(* CODESYS project CoDeSys PLC Program-Client.project

Project tree, tasks and I/O mapping:
  Device : CECC-LK, Festo AG & Co. KG, order no. 574418, version 3.5.0.7
    application Application
      libraries: Util, 3.5.0.0 (System); OPAK_RFID, 3.5.0.0 (elrest Automationssysteme GmbH); Solution Center Library, 3.5.8.0 (Festo Didactic SE - Customer Solution Center); Network, 3.5.7.0 (3S - Smart Software Solutions GmbH); Standard, 3.5.9.0 (System); Solution Center Library, 3.5.8.0 (Festo Didactic SE - Customer Solution Center); CAA CiA 405, 3.5.0.0 (CAA Technical Workgroup)
      task MainTask (cyclic, interval t#20ms, priority 20) calls PLC_PRG
      program PLC_PRG [ST]
      global variables IO
    Onboard : CECC 14I/8O, Festo AG & Co. KG, version 3.4.5.5
        unmapped channels: Onboard Input, Onboard Output
      Digital Inputs
          unmapped channels: Onboard Input
      Digital Outputs
          unmapped channels: Onboard Output
    CAN : CANbus, 3S - Smart Software Solutions GmbH, version 3.5.7.0
        settings: Baudrate = 1000
      CANopen : CANopen_Manager, 3S - Smart Software Solutions GmbH, order no. 1806, version 3.5.0.0
          settings: Sync CycleTime in Microseconds = 8000; Synchronous Window Length = 0; Enable Heartbeat generation = FALSE; CANopen NodeID = 1; ConfigVersion = 50659328
        BL20_GWBR_CANOPEN : BL20-GWBR-CANOPEN, TURCK, order no. 6827167, version Revision=16#00040017, FileVersion=4.23
            settings: General Options.Reset Node = FALSE; NODEIDSAVED = 2; SDO Timeout = 1000000; EXPERTSETTINGS = TRUE; Emergency-General Parameters.Emergency COBID = 16#82; Settings.COBID = 16#00000202; Settings.Transmission Type = 16#FF; Settings.available PDO-Parameter.Inhibit Time available = FALSE; Settings.available PDO-Parameter.Event Timer available = FALSE; Settings.Inhibit Time = 0; Settings.Event Timer = 0; Generic COBID = '$NODEID+16#0200'; Process by CANopenManager = TRUE; Settings.COBID = 16#00000302; Settings.Transmission Type = 16#FF; Settings.available PDO-Parameter.Inhibit Time available = FALSE; Settings.available PDO-Parameter.Event Timer available = FALSE; Settings.Inhibit Time = 0; Settings.Event Timer = 0; Generic COBID = '$NODEID+16#0300'; Process by CANopenManager = TRUE; Settings.COBID = 16#00000182; Settings.Transmission Type = 16#FF; Settings.available PDO-Parameter.Inhibit Time available = TRUE; Settings.available PDO-Parameter.Event Timer available = TRUE; Settings.Inhibit Time = 0; Settings.Event Timer = 0; Generic COBID = '$NODEID+16#0180'; Process by CANopenManager = TRUE; Settings.COBID = 16#00000282; Settings.Transmission Type = 16#FF; Settings.available PDO-Parameter.Inhibit Time available = TRUE; Settings.available PDO-Parameter.Event Timer available = TRUE; Settings.Inhibit Time = 0; Settings.Event Timer = 0; Generic COBID = '$NODEID+16#0280'; Process by CANopenManager = TRUE; WriteOutput8Bit : Generic_BL20_4DO.Index = 16#6200; WriteOutput8Bit : Generic_BL20_4DO.Subindex = 16#01; WriteOutput8Bit : Generic_BL20_4DO.ObjectLength = 8;
              WriteOutput8Bit : Generic_BL20_4DO_2.Index = 16#6200; WriteOutput8Bit : Generic_BL20_4DO_2.Subindex = 16#02; WriteOutput8Bit : Generic_BL20_4DO_2.ObjectLength = 8; WriteAnalogueOutput16 : Generic_BL20_2AO.Index = 16#6411; WriteAnalogueOutput16 : Generic_BL20_2AO.Subindex = 16#01; WriteAnalogueOutput16 : Generic_BL20_2AO.ObjectLength = 16; WriteAnalogueOutput16 : Generic_BL20_2AO.Index = 16#6411; WriteAnalogueOutput16 : Generic_BL20_2AO.Subindex = 16#02; WriteAnalogueOutput16 : Generic_BL20_2AO.ObjectLength = 16; ReadInput8Bit : Generic_BL20_4DI.Index = 16#6000; ReadInput8Bit : Generic_BL20_4DI.Subindex = 16#01; ReadInput8Bit : Generic_BL20_4DI.ObjectLength = 8; ReadAnalogueInput16Bit : Generic_BL20_4AI.Index = 16#6401; ReadAnalogueInput16Bit : Generic_BL20_4AI.Subindex = 16#01; ReadAnalogueInput16Bit : Generic_BL20_4AI.ObjectLength = 16; ReadAnalogueInput16Bit : Generic_BL20_4AI.Index = 16#6401; ReadAnalogueInput16Bit : Generic_BL20_4AI.Subindex = 16#02; ReadAnalogueInput16Bit : Generic_BL20_4AI.ObjectLength = 16; ReadAnalogueInput16Bit : Generic_BL20_4AI.Index = 16#6401; ReadAnalogueInput16Bit : Generic_BL20_4AI.Subindex = 16#03; ReadAnalogueInput16Bit : Generic_BL20_4AI.ObjectLength = 16; ReadAnalogueInput16Bit : Generic_BL20_4AI.Index = 16#6401; ReadAnalogueInput16Bit : Generic_BL20_4AI.Subindex = 16#04; ReadAnalogueInput16Bit : Generic_BL20_4AI.ObjectLength = 16; Number of SDO = 39; Set Guardtime.Index = 16#100C; Set Guardtime.Subindex = 16#00; Set Guardtime.Value = 16#00000000; Set Guardtime.Size = 16; Set Guardtime.AbortIfError = FALSE; Set Guardtime.JumpToLine = FALSE; Set Guardtime.Line = 0; Set Lifetime.Index = 16#100D; Set Lifetime.Subindex = 16#00; Set Lifetime.Value = 16#00000000; Set Lifetime.Size = 8; Set Lifetime.AbortIfError = FALSE; Set Lifetime.JumpToLine = FALSE; Set Lifetime.Line = 0; Disable Emcy CobID.Index = 16#1014;
              Disable Emcy CobID.Subindex = 16#00; Disable Emcy CobID.Value = 16#80000082; Disable Emcy CobID.Size = 32; Disable Emcy CobID.AbortIfError = FALSE; Disable Emcy CobID.JumpToLine = FALSE; Disable Emcy CobID.Line = 0; Set Emcy CobID.Index = 16#1014; Set Emcy CobID.Subindex = 16#00; Set Emcy CobID.Value = 16#00000082; Set Emcy CobID.Size = 32; Set Emcy CobID.AbortIfError = FALSE; Set Emcy CobID.JumpToLine = FALSE; Set Emcy CobID.Line = 0; Set Heartbeat Consumer.Index = 16#1016; Set Heartbeat Consumer.Subindex = 16#01; Set Heartbeat Consumer.Value = 0; Set Heartbeat Consumer.Size = 32; Set Heartbeat Consumer.AbortIfError = FALSE; Set Heartbeat Consumer.JumpToLine = FALSE; Set Heartbeat Consumer.Line = 0; Set Heartbeat Producer.Index = 16#1017; Set Heartbeat Producer.Subindex = 16#00; Set Heartbeat Producer.Value = 16#00000000; Set Heartbeat Producer.Size = 16; Set Heartbeat Producer.AbortIfError = FALSE; Set Heartbeat Producer.JumpToLine = FALSE; Set Heartbeat Producer.Line = 0; Disable PDO.Index = 16#1400; Disable PDO.Subindex = 16#01; Disable PDO.Value = 16#80000202; Disable PDO.Size = 32; Disable PDO.AbortIfError = FALSE; Disable PDO.JumpToLine = FALSE; Disable PDO.Line = 0; Set transmission type.Index = 16#1400; Set transmission type.Subindex = 16#02; Set transmission type.Value = 16#FF; Set transmission type.Size = 8; Set transmission type.AbortIfError = FALSE; Set transmission type.JumpToLine = FALSE;
              Set transmission type.Line = 0; Clear pdo mapping.Index = 16#1600; Clear pdo mapping.Subindex = 16#00; Clear pdo mapping.Value = 16#0; Clear pdo mapping.Size = 8; Clear pdo mapping.AbortIfError = FALSE; Clear pdo mapping.JumpToLine = FALSE; Clear pdo mapping.Line = 0; Set Mapping.Index = 16#1600; Set Mapping.Subindex = 16#01; Set Mapping.Value = 16#62000108; Set Mapping.Size = 32; Set Mapping.AbortIfError = FALSE; Set Mapping.JumpToLine = FALSE; Set Mapping.Line = 0; Set Mapping.Index = 16#1600; Set Mapping.Subindex = 16#02; Set Mapping.Value = 16#62000208; Set Mapping.Size = 32; Set Mapping.AbortIfError = FALSE; Set Mapping.JumpToLine = FALSE; Set Mapping.Line = 0; Set number of mappings.Index = 16#1600; Set number of mappings.Subindex = 16#00; Set number of mappings.Value = 16#02; Set number of mappings.Size = 8; Set number of mappings.AbortIfError = FALSE; Set number of mappings.JumpToLine = FALSE; Set number of mappings.Line = 0; Set and enable COB-ID.Index = 16#1400; Set and enable COB-ID.Subindex = 16#01; Set and enable COB-ID.Value = 16#00000202; Set and enable COB-ID.Size = 32; Set and enable COB-ID.AbortIfError = FALSE; Set and enable COB-ID.JumpToLine = FALSE; Set and enable COB-ID.Line = 0; Disable PDO.Index = 16#1401; Disable PDO.Subindex = 16#01; Disable PDO.Value = 16#80000302; Disable PDO.Size = 32;
              Disable PDO.AbortIfError = FALSE; Disable PDO.JumpToLine = FALSE; Disable PDO.Line = 0; Set transmission type.Index = 16#1401; Set transmission type.Subindex = 16#02; Set transmission type.Value = 16#FF; Set transmission type.Size = 8; Set transmission type.AbortIfError = FALSE; Set transmission type.JumpToLine = FALSE; Set transmission type.Line = 0; Clear pdo mapping.Index = 16#1601; Clear pdo mapping.Subindex = 16#00; Clear pdo mapping.Value = 16#0; Clear pdo mapping.Size = 8; Clear pdo mapping.AbortIfError = FALSE; Clear pdo mapping.JumpToLine = FALSE; Clear pdo mapping.Line = 0; Set Mapping.Index = 16#1601; Set Mapping.Subindex = 16#01; Set Mapping.Value = 16#64110110; Set Mapping.Size = 32; Set Mapping.AbortIfError = FALSE; Set Mapping.JumpToLine = FALSE; Set Mapping.Line = 0; Set Mapping.Index = 16#1601; Set Mapping.Subindex = 16#02; Set Mapping.Value = 16#64110210; Set Mapping.Size = 32; Set Mapping.AbortIfError = FALSE; Set Mapping.JumpToLine = FALSE; Set Mapping.Line = 0; Set number of mappings.Index = 16#1601; Set number of mappings.Subindex = 16#00; Set number of mappings.Value = 16#02; Set number of mappings.Size = 8; Set number of mappings.AbortIfError = FALSE; Set number of mappings.JumpToLine = FALSE; Set number of mappings.Line = 0; Set and enable COB-ID.Index = 16#1401; Set and enable COB-ID.Subindex = 16#01;
              Set and enable COB-ID.Value = 16#00000302; Set and enable COB-ID.Size = 32; Set and enable COB-ID.AbortIfError = FALSE; Set and enable COB-ID.JumpToLine = FALSE; Set and enable COB-ID.Line = 0; Disable PDO.Index = 16#1800; Disable PDO.Subindex = 16#01; Disable PDO.Value = 16#80000182; Disable PDO.Size = 32; Disable PDO.AbortIfError = FALSE; Disable PDO.JumpToLine = FALSE; Disable PDO.Line = 0; Set transmission type.Index = 16#1800; Set transmission type.Subindex = 16#02; Set transmission type.Value = 16#FF; Set transmission type.Size = 8; Set transmission type.AbortIfError = FALSE; Set transmission type.JumpToLine = FALSE; Set transmission type.Line = 0; Set inhibit time.Index = 16#1800; Set inhibit time.Subindex = 16#03; Set inhibit time.Value = 16#0000; Set inhibit time.Size = 16; Set inhibit time.AbortIfError = FALSE; Set inhibit time.JumpToLine = FALSE; Set inhibit time.Line = 0; Set event time.Index = 16#1800; Set event time.Subindex = 16#05; Set event time.Value = 16#0000; Set event time.Size = 16; Set event time.AbortIfError = FALSE; Set event time.JumpToLine = FALSE; Set event time.Line = 0; Clear pdo mapping.Index = 16#1A00; Clear pdo mapping.Subindex = 16#00; Clear pdo mapping.Value = 16#0; Clear pdo mapping.Size = 8; Clear pdo mapping.AbortIfError = FALSE; Clear pdo mapping.JumpToLine = FALSE; Clear pdo mapping.Line = 0;
              Set Mapping.Index = 16#1A00; Set Mapping.Subindex = 16#01; Set Mapping.Value = 16#60000108; Set Mapping.Size = 32; Set Mapping.AbortIfError = FALSE; Set Mapping.JumpToLine = FALSE; Set Mapping.Line = 0; Set number of mappings.Index = 16#1A00; Set number of mappings.Subindex = 16#00; Set number of mappings.Value = 16#01; Set number of mappings.Size = 8; Set number of mappings.AbortIfError = FALSE; Set number of mappings.JumpToLine = FALSE; Set number of mappings.Line = 0; Set and enable COB-ID.Index = 16#1800; Set and enable COB-ID.Subindex = 16#01; Set and enable COB-ID.Value = 16#00000182; Set and enable COB-ID.Size = 32; Set and enable COB-ID.AbortIfError = FALSE; Set and enable COB-ID.JumpToLine = FALSE; Set and enable COB-ID.Line = 0; Disable PDO.Index = 16#1801; Disable PDO.Subindex = 16#01; Disable PDO.Value = 16#80000282; Disable PDO.Size = 32; Disable PDO.AbortIfError = FALSE; Disable PDO.JumpToLine = FALSE; Disable PDO.Line = 0; Set transmission type.Index = 16#1801; Set transmission type.Subindex = 16#02; Set transmission type.Value = 16#FF; Set transmission type.Size = 8; Set transmission type.AbortIfError = FALSE; Set transmission type.JumpToLine = FALSE; Set transmission type.Line = 0; Set inhibit time.Index = 16#1801; Set inhibit time.Subindex = 16#03; Set inhibit time.Value = 16#0000; Set inhibit time.Size = 16; Set inhibit time.AbortIfError = FALSE;
              Set inhibit time.JumpToLine = FALSE; Set inhibit time.Line = 0; Set event time.Index = 16#1801; Set event time.Subindex = 16#05; Set event time.Value = 16#0000; Set event time.Size = 16; Set event time.AbortIfError = FALSE; Set event time.JumpToLine = FALSE; Set event time.Line = 0; Clear pdo mapping.Index = 16#1A01; Clear pdo mapping.Subindex = 16#00; Clear pdo mapping.Value = 16#0; Clear pdo mapping.Size = 8; Clear pdo mapping.AbortIfError = FALSE; Clear pdo mapping.JumpToLine = FALSE; Clear pdo mapping.Line = 0; Set Mapping.Index = 16#1A01; Set Mapping.Subindex = 16#01; Set Mapping.Value = 16#64010110; Set Mapping.Size = 32; Set Mapping.AbortIfError = FALSE; Set Mapping.JumpToLine = FALSE; Set Mapping.Line = 0; Set Mapping.Index = 16#1A01; Set Mapping.Subindex = 16#02; Set Mapping.Value = 16#64010210; Set Mapping.Size = 32; Set Mapping.AbortIfError = FALSE; Set Mapping.JumpToLine = FALSE; Set Mapping.Line = 0; Set Mapping.Index = 16#1A01; Set Mapping.Subindex = 16#03; Set Mapping.Value = 16#64010310; Set Mapping.Size = 32; Set Mapping.AbortIfError = FALSE; Set Mapping.JumpToLine = FALSE; Set Mapping.Line = 0; Set Mapping.Index = 16#1A01; Set Mapping.Subindex = 16#04; Set Mapping.Value = 16#64010410;
              Set Mapping.Size = 32; Set Mapping.AbortIfError = FALSE; Set Mapping.JumpToLine = FALSE; Set Mapping.Line = 0; Set number of mappings.Index = 16#1A01; Set number of mappings.Subindex = 16#00; Set number of mappings.Value = 16#04; Set number of mappings.Size = 8; Set number of mappings.AbortIfError = FALSE; Set number of mappings.JumpToLine = FALSE; Set number of mappings.Line = 0; Set and enable COB-ID.Index = 16#1801; Set and enable COB-ID.Subindex = 16#01; Set and enable COB-ID.Value = 16#00000282; Set and enable COB-ID.Size = 32; Set and enable COB-ID.AbortIfError = FALSE; Set and enable COB-ID.JumpToLine = FALSE; Set and enable COB-ID.Line = 0; ConfigVersion = 50659328
          Generic_BL20_4DI : Generic BL20-4DI, TURCK, order no. 0, version Revision=16#00040017, FileVersion=4.23
              settings: Number of Params = 0; Number of Params = 4; ReadInput8Bit : Generic_BL20_4DI.Index = 16#6000; ReadInput8Bit : Generic_BL20_4DI.Subindex = 16#01; ReadInput8Bit : Generic_BL20_4DI.Startbit = 0; ReadInput8Bit : Generic_BL20_4DI.Endbit = 0; ReadInput8Bit : Generic_BL20_4DI.Index = 16#6000; ReadInput8Bit : Generic_BL20_4DI.Subindex = 16#01; ReadInput8Bit : Generic_BL20_4DI.Startbit = 1; ReadInput8Bit : Generic_BL20_4DI.Endbit = 1; ReadInput8Bit : Generic_BL20_4DI.Index = 16#6000; ReadInput8Bit : Generic_BL20_4DI.Subindex = 16#01; ReadInput8Bit : Generic_BL20_4DI.Startbit = 2; ReadInput8Bit : Generic_BL20_4DI.Endbit = 2; ReadInput8Bit : Generic_BL20_4DI.Index = 16#6000; ReadInput8Bit : Generic_BL20_4DI.Subindex = 16#01; ReadInput8Bit : Generic_BL20_4DI.Startbit = 3; ReadInput8Bit : Generic_BL20_4DI.Endbit = 3
              unmapped channels: ReadInput8Bit : Generic_BL20_4DI, ReadInput8Bit : Generic_BL20_4DI, ReadInput8Bit : Generic_BL20_4DI, ReadInput8Bit : Generic_BL20_4DI
          Generic_BL20_4DI_1 : Generic BL20-4DI, TURCK, order no. 0, version Revision=16#00040017, FileVersion=4.23
              settings: Number of Params = 0; Number of Params = 4; ReadInput8Bit : Generic_BL20_4DI.Index = 16#6000; ReadInput8Bit : Generic_BL20_4DI.Subindex = 16#01; ReadInput8Bit : Generic_BL20_4DI.Startbit = 4; ReadInput8Bit : Generic_BL20_4DI.Endbit = 4; ReadInput8Bit : Generic_BL20_4DI.Index = 16#6000; ReadInput8Bit : Generic_BL20_4DI.Subindex = 16#01; ReadInput8Bit : Generic_BL20_4DI.Startbit = 5; ReadInput8Bit : Generic_BL20_4DI.Endbit = 5; ReadInput8Bit : Generic_BL20_4DI.Index = 16#6000; ReadInput8Bit : Generic_BL20_4DI.Subindex = 16#01; ReadInput8Bit : Generic_BL20_4DI.Startbit = 6; ReadInput8Bit : Generic_BL20_4DI.Endbit = 6; ReadInput8Bit : Generic_BL20_4DI.Index = 16#6000; ReadInput8Bit : Generic_BL20_4DI.Subindex = 16#01; ReadInput8Bit : Generic_BL20_4DI.Startbit = 7; ReadInput8Bit : Generic_BL20_4DI.Endbit = 7
              unmapped channels: ReadInput8Bit : Generic_BL20_4DI, ReadInput8Bit : Generic_BL20_4DI, ReadInput8Bit : Generic_BL20_4DI, ReadInput8Bit : Generic_BL20_4DI
          Generic_BL20_BR_PF : Generic BL20-BR/-PF, TURCK, order no. 0, version Revision=16#00040017, FileVersion=4.23
              settings: Number of Params = 0; Number of Params = 0
          Generic_BL20_4DO : Generic BL20-4DO, TURCK, order no. 0, version Revision=16#00040017, FileVersion=4.23
              settings: Number of Params = 4; WriteOutput8Bit : Generic_BL20_4DO.Index = 16#6200; WriteOutput8Bit : Generic_BL20_4DO.Subindex = 16#01; WriteOutput8Bit : Generic_BL20_4DO.Startbit = 0; WriteOutput8Bit : Generic_BL20_4DO.Endbit = 0; WriteOutput8Bit : Generic_BL20_4DO.Index = 16#6200; WriteOutput8Bit : Generic_BL20_4DO.Subindex = 16#01; WriteOutput8Bit : Generic_BL20_4DO.Startbit = 1; WriteOutput8Bit : Generic_BL20_4DO.Endbit = 1; WriteOutput8Bit : Generic_BL20_4DO.Index = 16#6200; WriteOutput8Bit : Generic_BL20_4DO.Subindex = 16#01; WriteOutput8Bit : Generic_BL20_4DO.Startbit = 2; WriteOutput8Bit : Generic_BL20_4DO.Endbit = 2; WriteOutput8Bit : Generic_BL20_4DO.Index = 16#6200; WriteOutput8Bit : Generic_BL20_4DO.Subindex = 16#01; WriteOutput8Bit : Generic_BL20_4DO.Startbit = 3; WriteOutput8Bit : Generic_BL20_4DO.Endbit = 3; Number of Params = 0
              unmapped channels: WriteOutput8Bit : Generic_BL20_4DO, WriteOutput8Bit : Generic_BL20_4DO, WriteOutput8Bit : Generic_BL20_4DO, WriteOutput8Bit : Generic_BL20_4DO
          Generic_BL20_4DO_1 : Generic BL20-4DO, TURCK, order no. 0, version Revision=16#00040017, FileVersion=4.23
              settings: Number of Params = 4; WriteOutput8Bit : Generic_BL20_4DO.Index = 16#6200; WriteOutput8Bit : Generic_BL20_4DO.Subindex = 16#01; WriteOutput8Bit : Generic_BL20_4DO.Startbit = 4; WriteOutput8Bit : Generic_BL20_4DO.Endbit = 4; WriteOutput8Bit : Generic_BL20_4DO.Index = 16#6200; WriteOutput8Bit : Generic_BL20_4DO.Subindex = 16#01; WriteOutput8Bit : Generic_BL20_4DO.Startbit = 5; WriteOutput8Bit : Generic_BL20_4DO.Endbit = 5; WriteOutput8Bit : Generic_BL20_4DO.Index = 16#6200; WriteOutput8Bit : Generic_BL20_4DO.Subindex = 16#01; WriteOutput8Bit : Generic_BL20_4DO.Startbit = 6; WriteOutput8Bit : Generic_BL20_4DO.Endbit = 6; WriteOutput8Bit : Generic_BL20_4DO.Index = 16#6200; WriteOutput8Bit : Generic_BL20_4DO.Subindex = 16#01; WriteOutput8Bit : Generic_BL20_4DO.Startbit = 7; WriteOutput8Bit : Generic_BL20_4DO.Endbit = 7; Number of Params = 0
              unmapped channels: WriteOutput8Bit : Generic_BL20_4DO, WriteOutput8Bit : Generic_BL20_4DO, WriteOutput8Bit : Generic_BL20_4DO, WriteOutput8Bit : Generic_BL20_4DO
          Generic_BL20_4DO_2 : Generic BL20-4DO, TURCK, order no. 0, version Revision=16#00040017, FileVersion=4.23
              settings: Number of Params = 4; WriteOutput8Bit : Generic_BL20_4DO_2.Index = 16#6200; WriteOutput8Bit : Generic_BL20_4DO_2.Subindex = 16#02; WriteOutput8Bit : Generic_BL20_4DO_2.Startbit = 0; WriteOutput8Bit : Generic_BL20_4DO_2.Endbit = 0; WriteOutput8Bit : Generic_BL20_4DO_2.Index = 16#6200; WriteOutput8Bit : Generic_BL20_4DO_2.Subindex = 16#02; WriteOutput8Bit : Generic_BL20_4DO_2.Startbit = 1; WriteOutput8Bit : Generic_BL20_4DO_2.Endbit = 1; WriteOutput8Bit : Generic_BL20_4DO_2.Index = 16#6200; WriteOutput8Bit : Generic_BL20_4DO_2.Subindex = 16#02; WriteOutput8Bit : Generic_BL20_4DO_2.Startbit = 2; WriteOutput8Bit : Generic_BL20_4DO_2.Endbit = 2; WriteOutput8Bit : Generic_BL20_4DO_2.Index = 16#6200; WriteOutput8Bit : Generic_BL20_4DO_2.Subindex = 16#02; WriteOutput8Bit : Generic_BL20_4DO_2.Startbit = 3; WriteOutput8Bit : Generic_BL20_4DO_2.Endbit = 3; Number of Params = 0
              unmapped channels: WriteOutput8Bit : Generic_BL20_4DO_2, WriteOutput8Bit : Generic_BL20_4DO_2, WriteOutput8Bit : Generic_BL20_4DO_2, WriteOutput8Bit : Generic_BL20_4DO_2
          Generic_BL20_4DO_3 : Generic BL20-4DO, TURCK, order no. 0, version Revision=16#00040017, FileVersion=4.23
              settings: Number of Params = 4; WriteOutput8Bit : Generic_BL20_4DO_2.Index = 16#6200; WriteOutput8Bit : Generic_BL20_4DO_2.Subindex = 16#02; WriteOutput8Bit : Generic_BL20_4DO_2.Startbit = 4; WriteOutput8Bit : Generic_BL20_4DO_2.Endbit = 4; WriteOutput8Bit : Generic_BL20_4DO_2.Index = 16#6200; WriteOutput8Bit : Generic_BL20_4DO_2.Subindex = 16#02; WriteOutput8Bit : Generic_BL20_4DO_2.Startbit = 5; WriteOutput8Bit : Generic_BL20_4DO_2.Endbit = 5; WriteOutput8Bit : Generic_BL20_4DO_2.Index = 16#6200; WriteOutput8Bit : Generic_BL20_4DO_2.Subindex = 16#02; WriteOutput8Bit : Generic_BL20_4DO_2.Startbit = 6; WriteOutput8Bit : Generic_BL20_4DO_2.Endbit = 6; WriteOutput8Bit : Generic_BL20_4DO_2.Index = 16#6200; WriteOutput8Bit : Generic_BL20_4DO_2.Subindex = 16#02; WriteOutput8Bit : Generic_BL20_4DO_2.Startbit = 7; WriteOutput8Bit : Generic_BL20_4DO_2.Endbit = 7; Number of Params = 0
              unmapped channels: WriteOutput8Bit : Generic_BL20_4DO_2, WriteOutput8Bit : Generic_BL20_4DO_2, WriteOutput8Bit : Generic_BL20_4DO_2, WriteOutput8Bit : Generic_BL20_4DO_2
          Generic_BL20_2AO : Generic BL20-2AO, TURCK, order no. 0, version Revision=16#00040017, FileVersion=4.23
              settings: Number of Params = 2; WriteAnalogueOutput16 : Generic_BL20_2AO.Index = 16#6411; WriteAnalogueOutput16 : Generic_BL20_2AO.Subindex = 16#01; WriteAnalogueOutput16 : Generic_BL20_2AO.Startbit = 0; WriteAnalogueOutput16 : Generic_BL20_2AO.Endbit = 15; WriteAnalogueOutput16 : Generic_BL20_2AO.Index = 16#6411; WriteAnalogueOutput16 : Generic_BL20_2AO.Subindex = 16#02; WriteAnalogueOutput16 : Generic_BL20_2AO.Startbit = 0; WriteAnalogueOutput16 : Generic_BL20_2AO.Endbit = 15; Number of Params = 0
              unmapped channels: WriteAnalogueOutput16 : Generic_BL20_2AO, WriteAnalogueOutput16 : Generic_BL20_2AO
          Generic_BL20_4AI : Generic BL20-4AI, TURCK, order no. 0, version Revision=16#00040017, FileVersion=4.23
              settings: Number of Params = 0; Number of Params = 4; ReadAnalogueInput16Bit : Generic_BL20_4AI.Index = 16#6401; ReadAnalogueInput16Bit : Generic_BL20_4AI.Subindex = 16#01; ReadAnalogueInput16Bit : Generic_BL20_4AI.Startbit = 0; ReadAnalogueInput16Bit : Generic_BL20_4AI.Endbit = 15; ReadAnalogueInput16Bit : Generic_BL20_4AI.Index = 16#6401; ReadAnalogueInput16Bit : Generic_BL20_4AI.Subindex = 16#02; ReadAnalogueInput16Bit : Generic_BL20_4AI.Startbit = 0; ReadAnalogueInput16Bit : Generic_BL20_4AI.Endbit = 15; ReadAnalogueInput16Bit : Generic_BL20_4AI.Index = 16#6401; ReadAnalogueInput16Bit : Generic_BL20_4AI.Subindex = 16#03; ReadAnalogueInput16Bit : Generic_BL20_4AI.Startbit = 0; ReadAnalogueInput16Bit : Generic_BL20_4AI.Endbit = 15; ReadAnalogueInput16Bit : Generic_BL20_4AI.Index = 16#6401; ReadAnalogueInput16Bit : Generic_BL20_4AI.Subindex = 16#04; ReadAnalogueInput16Bit : Generic_BL20_4AI.Startbit = 0; ReadAnalogueInput16Bit : Generic_BL20_4AI.Endbit = 15
              unmapped channels: ReadAnalogueInput16Bit : Generic_BL20_4AI, ReadAnalogueInput16Bit : Generic_BL20_4AI, ReadAnalogueInput16Bit : Generic_BL20_4AI, ReadAnalogueInput16Bit : Generic_BL20_4AI
        DTM425 : DTM425, ifm electronic gmbh, order no. DTM425, version Revision=16#00000000, FileVersion=8.2
            settings: General Options.Reset Node = FALSE; NODEIDSAVED = 32; SDO Timeout = 1000000; EXPERTSETTINGS = TRUE; Emergency-General Parameters.Emergency COBID = 16#A0; PDO 16#1400.COBID = 16#00000220; Process by CANopenManager = TRUE; PDO 16#1401.COBID = 16#00000320; Process by CANopenManager = TRUE; PDO 16#1402.COBID = 16#00000420; Process by CANopenManager = TRUE; PDO 16#1403.COBID = 16#00000520; Process by CANopenManager = TRUE; PDO 16#1800.COBID = 16#000001A0; PDO 16#1800.Event Timer = 0; Process by CANopenManager = TRUE; PDO 16#1801.COBID = 16#000002A0; PDO 16#1801.Event Timer = 0; Process by CANopenManager = TRUE; PDO 16#1802.COBID = 16#000003A0; PDO 16#1802.Event Timer = 0; Process by CANopenManager = TRUE; PDO 16#1803.COBID = 16#000004A0; PDO 16#1803.Event Timer = 0; Process by CANopenManager = TRUE; Write Data (mappable): Write Trigger.Subindex = 16#00; Write Data (mappable): Data_sub1.Subindex = 16#01; Write Data (mappable): Data_sub2.Subindex = 16#02; Write Data (mappable): Data_sub3.Subindex = 16#03; Device Status.Subindex = 16#00; Read Data (mappable): Data_sub1.Subindex = 16#01; Read Data (mappable): Data_sub2.Subindex = 16#02; Read Data (mappable): Data_sub3.Subindex = 16#03; Number of SDO = 55; Disable Emcy CobID.Index = 16#1014; Disable Emcy CobID.Subindex = 16#00; Disable Emcy CobID.Value = 16#800000A0; Disable Emcy CobID.Size = 32; Disable Emcy CobID.AbortIfError = FALSE; Disable Emcy CobID.JumpToLine = FALSE;
              Disable Emcy CobID.Line = 0; Set Emcy CobID.Index = 16#1014; Set Emcy CobID.Subindex = 16#00; Set Emcy CobID.Value = 16#000000A0; Set Emcy CobID.Size = 32; Set Emcy CobID.AbortIfError = FALSE; Set Emcy CobID.JumpToLine = FALSE; Set Emcy CobID.Line = 0; Set Heartbeat Producer.Index = 16#1017; Set Heartbeat Producer.Subindex = 16#00; Set Heartbeat Producer.Value = 16#00000000; Set Heartbeat Producer.Size = 16; Set Heartbeat Producer.AbortIfError = FALSE; Set Heartbeat Producer.JumpToLine = FALSE; Set Heartbeat Producer.Line = 0; Disable PDO.Index = 16#1400; Disable PDO.Subindex = 16#01; Disable PDO.Value = 16#80000220; Disable PDO.Size = 32; Disable PDO.AbortIfError = FALSE; Disable PDO.JumpToLine = FALSE; Disable PDO.Line = 0; Set transmission type.Index = 16#1400; Set transmission type.Subindex = 16#02; Set transmission type.Value = 16#FF; Set transmission type.Size = 8; Set transmission type.AbortIfError = FALSE; Set transmission type.JumpToLine = FALSE; Set transmission type.Line = 0; Clear pdo mapping.Index = 16#1600; Clear pdo mapping.Subindex = 16#00; Clear pdo mapping.Value = 16#0; Clear pdo mapping.Size = 8; Clear pdo mapping.AbortIfError = FALSE; Clear pdo mapping.JumpToLine = FALSE; Clear pdo mapping.Line = 0; Set Mapping.Index = 16#1600; Set Mapping.Subindex = 16#01; Set Mapping.Value = 16#230F0040; Set Mapping.Size = 32;
              Set Mapping.AbortIfError = FALSE; Set Mapping.JumpToLine = FALSE; Set Mapping.Line = 0; Set number of mappings.Index = 16#1600; Set number of mappings.Subindex = 16#00; Set number of mappings.Value = 16#01; Set number of mappings.Size = 8; Set number of mappings.AbortIfError = FALSE; Set number of mappings.JumpToLine = FALSE; Set number of mappings.Line = 0; Set and enable COB-ID.Index = 16#1400; Set and enable COB-ID.Subindex = 16#01; Set and enable COB-ID.Value = 16#00000220; Set and enable COB-ID.Size = 32; Set and enable COB-ID.AbortIfError = FALSE; Set and enable COB-ID.JumpToLine = FALSE; Set and enable COB-ID.Line = 0; Disable PDO.Index = 16#1401; Disable PDO.Subindex = 16#01; Disable PDO.Value = 16#80000320; Disable PDO.Size = 32; Disable PDO.AbortIfError = FALSE; Disable PDO.JumpToLine = FALSE; Disable PDO.Line = 0; Set transmission type.Index = 16#1401; Set transmission type.Subindex = 16#02; Set transmission type.Value = 16#FF; Set transmission type.Size = 8; Set transmission type.AbortIfError = FALSE; Set transmission type.JumpToLine = FALSE; Set transmission type.Line = 0; Clear pdo mapping.Index = 16#1601; Clear pdo mapping.Subindex = 16#00; Clear pdo mapping.Value = 16#0; Clear pdo mapping.Size = 8; Clear pdo mapping.AbortIfError = FALSE; Clear pdo mapping.JumpToLine = FALSE; Clear pdo mapping.Line = 0; Set Mapping.Index = 16#1601; Set Mapping.Subindex = 16#01;
              Set Mapping.Value = 16#230A0140; Set Mapping.Size = 32; Set Mapping.AbortIfError = FALSE; Set Mapping.JumpToLine = FALSE; Set Mapping.Line = 0; Set number of mappings.Index = 16#1601; Set number of mappings.Subindex = 16#00; Set number of mappings.Value = 16#01; Set number of mappings.Size = 8; Set number of mappings.AbortIfError = FALSE; Set number of mappings.JumpToLine = FALSE; Set number of mappings.Line = 0; Set and enable COB-ID.Index = 16#1401; Set and enable COB-ID.Subindex = 16#01; Set and enable COB-ID.Value = 16#00000320; Set and enable COB-ID.Size = 32; Set and enable COB-ID.AbortIfError = FALSE; Set and enable COB-ID.JumpToLine = FALSE; Set and enable COB-ID.Line = 0; Disable PDO.Index = 16#1402; Disable PDO.Subindex = 16#01; Disable PDO.Value = 16#80000420; Disable PDO.Size = 32; Disable PDO.AbortIfError = FALSE; Disable PDO.JumpToLine = FALSE; Disable PDO.Line = 0; Set transmission type.Index = 16#1402; Set transmission type.Subindex = 16#02; Set transmission type.Value = 16#FF; Set transmission type.Size = 8; Set transmission type.AbortIfError = FALSE; Set transmission type.JumpToLine = FALSE; Set transmission type.Line = 0; Clear pdo mapping.Index = 16#1602; Clear pdo mapping.Subindex = 16#00; Clear pdo mapping.Value = 16#0; Clear pdo mapping.Size = 8; Clear pdo mapping.AbortIfError = FALSE; Clear pdo mapping.JumpToLine = FALSE; Clear pdo mapping.Line = 0;
              Set Mapping.Index = 16#1602; Set Mapping.Subindex = 16#01; Set Mapping.Value = 16#230A0240; Set Mapping.Size = 32; Set Mapping.AbortIfError = FALSE; Set Mapping.JumpToLine = FALSE; Set Mapping.Line = 0; Set number of mappings.Index = 16#1602; Set number of mappings.Subindex = 16#00; Set number of mappings.Value = 16#01; Set number of mappings.Size = 8; Set number of mappings.AbortIfError = FALSE; Set number of mappings.JumpToLine = FALSE; Set number of mappings.Line = 0; Set and enable COB-ID.Index = 16#1402; Set and enable COB-ID.Subindex = 16#01; Set and enable COB-ID.Value = 16#00000420; Set and enable COB-ID.Size = 32; Set and enable COB-ID.AbortIfError = FALSE; Set and enable COB-ID.JumpToLine = FALSE; Set and enable COB-ID.Line = 0; Disable PDO.Index = 16#1403; Disable PDO.Subindex = 16#01; Disable PDO.Value = 16#80000520; Disable PDO.Size = 32; Disable PDO.AbortIfError = FALSE; Disable PDO.JumpToLine = FALSE; Disable PDO.Line = 0; Set transmission type.Index = 16#1403; Set transmission type.Subindex = 16#02; Set transmission type.Value = 16#FF; Set transmission type.Size = 8; Set transmission type.AbortIfError = FALSE; Set transmission type.JumpToLine = FALSE; Set transmission type.Line = 0; Clear pdo mapping.Index = 16#1603; Clear pdo mapping.Subindex = 16#00; Clear pdo mapping.Value = 16#0; Clear pdo mapping.Size = 8; Clear pdo mapping.AbortIfError = FALSE;
              Clear pdo mapping.JumpToLine = FALSE; Clear pdo mapping.Line = 0; Set Mapping.Index = 16#1603; Set Mapping.Subindex = 16#01; Set Mapping.Value = 16#230A0340; Set Mapping.Size = 32; Set Mapping.AbortIfError = FALSE; Set Mapping.JumpToLine = FALSE; Set Mapping.Line = 0; Set number of mappings.Index = 16#1603; Set number of mappings.Subindex = 16#00; Set number of mappings.Value = 16#01; Set number of mappings.Size = 8; Set number of mappings.AbortIfError = FALSE; Set number of mappings.JumpToLine = FALSE; Set number of mappings.Line = 0; Set and enable COB-ID.Index = 16#1403; Set and enable COB-ID.Subindex = 16#01; Set and enable COB-ID.Value = 16#00000520; Set and enable COB-ID.Size = 32; Set and enable COB-ID.AbortIfError = FALSE; Set and enable COB-ID.JumpToLine = FALSE; Set and enable COB-ID.Line = 0; Disable PDO.Index = 16#1800; Disable PDO.Subindex = 16#01; Disable PDO.Value = 16#800001A0; Disable PDO.Size = 32; Disable PDO.AbortIfError = FALSE; Disable PDO.JumpToLine = FALSE; Disable PDO.Line = 0; Set transmission type.Index = 16#1800; Set transmission type.Subindex = 16#02; Set transmission type.Value = 16#FF; Set transmission type.Size = 8; Set transmission type.AbortIfError = FALSE; Set transmission type.JumpToLine = FALSE; Set transmission type.Line = 0; Set inhibit time.Index = 16#1800; Set inhibit time.Subindex = 16#03; Set inhibit time.Value = 16#00C8;
              Set inhibit time.Size = 16; Set inhibit time.AbortIfError = FALSE; Set inhibit time.JumpToLine = FALSE; Set inhibit time.Line = 0; Clear pdo mapping.Index = 16#1A00; Clear pdo mapping.Subindex = 16#00; Clear pdo mapping.Value = 16#0; Clear pdo mapping.Size = 8; Clear pdo mapping.AbortIfError = FALSE; Clear pdo mapping.JumpToLine = FALSE; Clear pdo mapping.Line = 0; Set Mapping.Index = 16#1A00; Set Mapping.Subindex = 16#01; Set Mapping.Value = 16#21500020; Set Mapping.Size = 32; Set Mapping.AbortIfError = FALSE; Set Mapping.JumpToLine = FALSE; Set Mapping.Line = 0; Set number of mappings.Index = 16#1A00; Set number of mappings.Subindex = 16#00; Set number of mappings.Value = 16#01; Set number of mappings.Size = 8; Set number of mappings.AbortIfError = FALSE; Set number of mappings.JumpToLine = FALSE; Set number of mappings.Line = 0; Set and enable COB-ID.Index = 16#1800; Set and enable COB-ID.Subindex = 16#01; Set and enable COB-ID.Value = 16#000001A0; Set and enable COB-ID.Size = 32; Set and enable COB-ID.AbortIfError = FALSE; Set and enable COB-ID.JumpToLine = FALSE; Set and enable COB-ID.Line = 0; Disable PDO.Index = 16#1801; Disable PDO.Subindex = 16#01; Disable PDO.Value = 16#800002A0; Disable PDO.Size = 32; Disable PDO.AbortIfError = FALSE; Disable PDO.JumpToLine = FALSE; Disable PDO.Line = 0; Set transmission type.Index = 16#1801;
              Set transmission type.Subindex = 16#02; Set transmission type.Value = 16#FF; Set transmission type.Size = 8; Set transmission type.AbortIfError = FALSE; Set transmission type.JumpToLine = FALSE; Set transmission type.Line = 0; Set inhibit time.Index = 16#1801; Set inhibit time.Subindex = 16#03; Set inhibit time.Value = 16#00C8; Set inhibit time.Size = 16; Set inhibit time.AbortIfError = FALSE; Set inhibit time.JumpToLine = FALSE; Set inhibit time.Line = 0; Clear pdo mapping.Index = 16#1A01; Clear pdo mapping.Subindex = 16#00; Clear pdo mapping.Value = 16#0; Clear pdo mapping.Size = 8; Clear pdo mapping.AbortIfError = FALSE; Clear pdo mapping.JumpToLine = FALSE; Clear pdo mapping.Line = 0; Set Mapping.Index = 16#1A01; Set Mapping.Subindex = 16#01; Set Mapping.Value = 16#220A0140; Set Mapping.Size = 32; Set Mapping.AbortIfError = FALSE; Set Mapping.JumpToLine = FALSE; Set Mapping.Line = 0; Set number of mappings.Index = 16#1A01; Set number of mappings.Subindex = 16#00; Set number of mappings.Value = 16#01; Set number of mappings.Size = 8; Set number of mappings.AbortIfError = FALSE; Set number of mappings.JumpToLine = FALSE; Set number of mappings.Line = 0; Set and enable COB-ID.Index = 16#1801; Set and enable COB-ID.Subindex = 16#01; Set and enable COB-ID.Value = 16#000002A0; Set and enable COB-ID.Size = 32; Set and enable COB-ID.AbortIfError = FALSE; Set and enable COB-ID.JumpToLine = FALSE;
              Set and enable COB-ID.Line = 0; Disable PDO.Index = 16#1802; Disable PDO.Subindex = 16#01; Disable PDO.Value = 16#800003A0; Disable PDO.Size = 32; Disable PDO.AbortIfError = FALSE; Disable PDO.JumpToLine = FALSE; Disable PDO.Line = 0; Set transmission type.Index = 16#1802; Set transmission type.Subindex = 16#02; Set transmission type.Value = 16#FF; Set transmission type.Size = 8; Set transmission type.AbortIfError = FALSE; Set transmission type.JumpToLine = FALSE; Set transmission type.Line = 0; Set inhibit time.Index = 16#1802; Set inhibit time.Subindex = 16#03; Set inhibit time.Value = 16#00C8; Set inhibit time.Size = 16; Set inhibit time.AbortIfError = FALSE; Set inhibit time.JumpToLine = FALSE; Set inhibit time.Line = 0; Clear pdo mapping.Index = 16#1A02; Clear pdo mapping.Subindex = 16#00; Clear pdo mapping.Value = 16#0; Clear pdo mapping.Size = 8; Clear pdo mapping.AbortIfError = FALSE; Clear pdo mapping.JumpToLine = FALSE; Clear pdo mapping.Line = 0; Set Mapping.Index = 16#1A02; Set Mapping.Subindex = 16#01; Set Mapping.Value = 16#220A0240; Set Mapping.Size = 32; Set Mapping.AbortIfError = FALSE; Set Mapping.JumpToLine = FALSE; Set Mapping.Line = 0; Set number of mappings.Index = 16#1A02; Set number of mappings.Subindex = 16#00; Set number of mappings.Value = 16#01; Set number of mappings.Size = 8;
              Set number of mappings.AbortIfError = FALSE; Set number of mappings.JumpToLine = FALSE; Set number of mappings.Line = 0; Set and enable COB-ID.Index = 16#1802; Set and enable COB-ID.Subindex = 16#01; Set and enable COB-ID.Value = 16#000003A0; Set and enable COB-ID.Size = 32; Set and enable COB-ID.AbortIfError = FALSE; Set and enable COB-ID.JumpToLine = FALSE; Set and enable COB-ID.Line = 0; Disable PDO.Index = 16#1803; Disable PDO.Subindex = 16#01; Disable PDO.Value = 16#800004A0; Disable PDO.Size = 32; Disable PDO.AbortIfError = FALSE; Disable PDO.JumpToLine = FALSE; Disable PDO.Line = 0; Set transmission type.Index = 16#1803; Set transmission type.Subindex = 16#02; Set transmission type.Value = 16#FF; Set transmission type.Size = 8; Set transmission type.AbortIfError = FALSE; Set transmission type.JumpToLine = FALSE; Set transmission type.Line = 0; Set inhibit time.Index = 16#1803; Set inhibit time.Subindex = 16#03; Set inhibit time.Value = 16#00C8; Set inhibit time.Size = 16; Set inhibit time.AbortIfError = FALSE; Set inhibit time.JumpToLine = FALSE; Set inhibit time.Line = 0; Clear pdo mapping.Index = 16#1A03; Clear pdo mapping.Subindex = 16#00; Clear pdo mapping.Value = 16#0; Clear pdo mapping.Size = 8; Clear pdo mapping.AbortIfError = FALSE; Clear pdo mapping.JumpToLine = FALSE; Clear pdo mapping.Line = 0; Set Mapping.Index = 16#1A03; Set Mapping.Subindex = 16#01;
              Set Mapping.Value = 16#220A0340; Set Mapping.Size = 32; Set Mapping.AbortIfError = FALSE; Set Mapping.JumpToLine = FALSE; Set Mapping.Line = 0; Set number of mappings.Index = 16#1A03; Set number of mappings.Subindex = 16#00; Set number of mappings.Value = 16#01; Set number of mappings.Size = 8; Set number of mappings.AbortIfError = FALSE; Set number of mappings.JumpToLine = FALSE; Set number of mappings.Line = 0; Set and enable COB-ID.Index = 16#1803; Set and enable COB-ID.Subindex = 16#01; Set and enable COB-ID.Value = 16#000004A0; Set and enable COB-ID.Size = 32; Set and enable COB-ID.AbortIfError = FALSE; Set and enable COB-ID.JumpToLine = FALSE; Set and enable COB-ID.Line = 0; ConfigVersion = 50659328
            unmapped channels: Write Data (mappable): Write Trigger, Write Data (mappable): Data_sub1, Write Data (mappable): Data_sub2, Write Data (mappable): Data_sub3, Device Status, Read Data (mappable): Data_sub1, Read Data (mappable): Data_sub2, Read Data (mappable): Data_sub3
*)

// Device/Application/IO
VAR_GLOBAL
	
	xBG20		AT %IX1.0	: BOOL;	// Stopper released
	xBG21		AT %IX1.1	: BOOL;	// Carrier available
	xBG22		AT %IX1.2	: BOOL;	// Carrier ID bit 0
	xBG23		AT %IX1.3	: BOOL;	// Carrier ID bit 1
	xBG24		AT %IX1.4	: BOOL;	// Carrier ID bit 2
	xEmg		AT %IX0.0	: BOOL;	// Emergency stop
	
	
	xMB20		AT %QX1.0	: BOOL;	// Release stopper
	xQA1_LEFT	AT %QX0.5	: BOOL;	// Conveyor to the left
	xQA1_RIGHT	AT %QX0.4	: BOOL;	// Conveyor to the right
	xQA1_SLOW	AT %QX0.6	: BOOL;	// Conveyor Slow
	xQA1_STOP	AT %QX0.7	: BOOL;	// Conveyor Stop
END_VAR

// Device/Application/PLC_PRG
PROGRAM PLC_PRG
VAR
	state			:	INT := 0 ;
	timer			:	TON;
	RFID			:	dc_ecp.Dtm425;
	rfidData		:	dc_ecp.st_CPF_RfidData;
	carrierID		: UINT;
	TCPclient		: dc_ecp.TcpClientByteStream;
	DataOUT			: DWORD;
	DataIN			: DWORD;
	XMLstring		: STRING;
	prcsDelay		: TIME;
	stationID		: UINT;
	DateTime		: STRING;
END_VAR

timer();
RFID();
TCPclient();

CASE state OF
	0: // Initialize
	IO.xQA1_RIGHT := TRUE;
	IO.xMB20 := FALSE;
	state := 1;
	
	1: // Connect RFID and TCPclient
	IF RFID.xReady THEN 
		RFID.Connect(usiNodeId := 32, usiNetworkId := 0, usiChannel := 1);
		TCPclient.Connect(sIP := 'localhost', uiPort := 40000);
		state := 2;
	END_IF
	
	2: // Check that RFID and TCPclient is ready and connected
	IF RFID.xReady AND TCPclient.xConnected AND TCPclient.xReady THEN
		state := 3;
	END_IF
	
	3: // Slow down conveyer belt before stop
	IO.xMB20 := FALSE;
	IF IO.xBG24 = TRUE THEN
		IO.xQA1_SLOW := TRUE;
		state := 4;
	END_IF
	
	4: // Read Data and Process
	IF IO.xBG21 = TRUE THEN
		rfid.ReadTag(uiStartAddress:=0,uiDataLength:=SIZEOF(rfidData), pData:=ADR(rfidData));
		carrierID:=dc_ecp.SwapWORD(rfidData.uiCarrierID); 	// Read out carrier-id
		stationID := 0; 									// Read station ID
		DateTime := '11/3/2020 16:20:42:11'; 				// Read current data and time
		XMLstring := '<carrierID>';							// Create XML string from data
		XMLstring := CONCAT(XMLstring, UINT_TO_STRING(carrierID));
		XMLstring := CONCAT(XMLstring, '<\carrierID>$N<stationID>');
		XMLstring := CONCAT(XMLstring, UINT_TO_STRING(stationID));
		XMLstring := CONCAT(XMLstring, '<\stationID>$N<DateTime>');
		XMLstring := CONCAT(XMLstring, DateTime);
		XMLstring := CONCAT(XMLstring, '<\DateTime>');
		state := 5;
	END_IF
	
	5: //
	IF IO.xBG21 = TRUE THEN 
		TCPclient.Send(pToSend := ADR(DataOUT), uiSizeToSend := SIZEOF(DataOUT));
		TCPclient.Receive(pToReceive := ADR(DataIN), uiSizeToReceive := SIZEOF(DataIN));
		
		prcsDelay := T#3S; // Processing Time 
		timer(IN:=TRUE,PT:=prcsDelay); // Wait for Proccesing Time before stopper release
		IF timer.Q = TRUE THEN
			timer.IN := FALSE;
			IO.xMB20 := TRUE;
			state := 6;
		END_IF
	END_IF
 
	6: //
	timer(IN:=TRUE,PT:=T#2S);	
	IF timer.Q = TRUE THEN
		timer.IN := FALSE;
		IO.xQA1_SLOW := FALSE;
		state := 1;
	END_IF
END_CASE

END_PROGRAM
